// TwinCAT 3 PLC project Plc
// ProgramVersion: 3.1.4024.0
// libraries:
//   Tc2_Standard, * (Beckhoff Automation GmbH)
//   Tc2_System, * (Beckhoff Automation GmbH)
//   Tc3_Module, * (Beckhoff Automation GmbH)
//   VisuSymbols,3.5.10.0,System
// project tree:
//   / Gestore di visualizzazione.TcVMO (not stored), GlobalTextList.TcGTLO, PlcTask.TcTTO
//   POUs/ MAIN.TcPOU
//   VISUs/ Visualization.TcVIS
// real-time tasks:
//   TASK PlcTask: cycle T#10ms, priority 20, ADS port 350

CONFIGURATION Plc
    RESOURCE PLC ON TwinCAT3
        TASK PlcTask(INTERVAL := T#10ms, PRIORITY := 20);
        PROGRAM MAIN WITH PlcTask : MAIN;
    END_RESOURCE
END_CONFIGURATION

// ---- POUs/MAIN.TcPOU
PROGRAM MAIN
VAR
	PBSTart: BOOL;
	PBStop: BOOL;
	Motor: BOOL;
END_VAR

IF PBSTop THEN
	Motor:= FALSE;
ELSIF PBSTart THEN
	Motor:= TRUE;
END_IF

END_PROGRAM

// ---- GlobalTextList.TcGTLO
TEXTLIST GlobalTextList
  10 = 'Start'
  123 = 'Stop'
  576 = 'Testo'
END_TEXTLIST

// ---- VISUs/Visualization.TcVIS
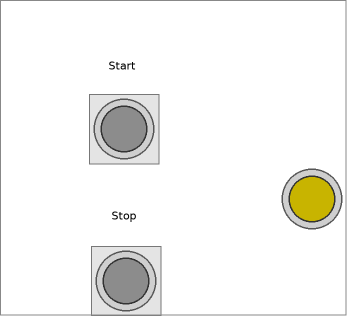
VISUALIZATION Visualization  // 347x316
    Lamp1 (277,164 70x70), variable: MAIN.Motor, style: Lamp-Lamp1-Yellow
    PushSwitch (89,94 70x70), variable: MAIN.PBSTart, behaviour: TAP, style: Switch-PushSwitch-Gray
    PushSwitch (91,246 70x70), variable: MAIN.PBStop, behaviour: TAP, style: Switch-PushSwitch-Gray
    Label (47,51 150x30), "Start"
    Label (49,201 150x30), "Stop"
END_VISUALIZATION
